TYPE TValve :
STRUCT
	Cmd : TValveCmd;
	State : TValveState;
	Time2Open : TIME := T#12S;
	
	OpenFailTimer : TON;
	CloseFailTimer : TON;
	
END_STRUCT
END_TYPE

(* stored: Version 1.1.0.1, ProductVersion 3.1.4024.13
   DUT TValve: Id {c769af80-eeba-4af4-9934-db9b2e751452} *)
